TYPE SequenceInfo :
STRUCT
	MoverId : UDINT;
	CurrentStation : INT;
	Velocity : MC_LREAL;
	State : StationSequenceState;
END_STRUCT
END_TYPE

(* stored: Version 1.1.0.1
   DUT SequenceInfo: Id {e31e4eaf-6c71-46bd-8e49-86316a781b98} *)
